// Mitsubishi GX Works2 project: ror_rorEx02   PLC: Q02/Q02H

PROGRAM MAIN
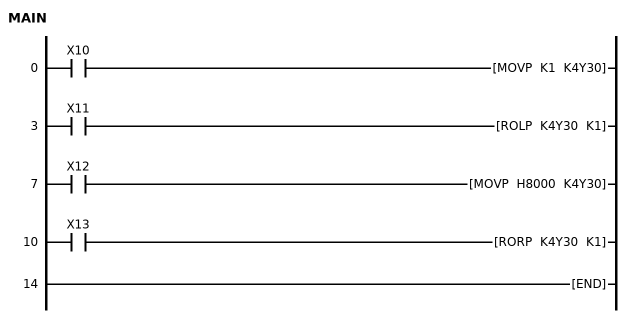
0     LD      X10
      MOVP    K1 K4Y30
3     LD      X11
      ROLP    K4Y30 K1
7     LD      X12
      MOVP    H8000 K4Y30
10    LD      X13
      RORP    K4Y30 K1
14    END
END_PROGRAM
